// TIA Portal project "2022.04.30-电机顺启" (V17)

(* hardware
DEVICE "S7-1500/ET200MP station_1"  S7-1500 station
   slot 0: "导轨_0"  Rack  6ES7 590-1***0-0AA0
   slot 1: "PLC_1"  CPU 1516-3 PN/DP  6ES7 516-3AN00-0AB0  V1.7
      slot 3: "CPU 显示_1"  6ES7591-1BA00-0AA0
      slot 32768: "PROFINET 接口_1"  X1
         slot 32769: "端口_1"  X1 P1
         slot 32770: "端口_2"  X1 P2
      slot 33024: "PROFINET 接口_2"  X2
         slot 33025: "端口_1"  X2 P1
      slot 33280: "DP 接口_1"  X3
   slot 2: "DI 32x24VDC BA_1"  DI 32x24VDC BA  6ES7 521-1BL10-0AA0  V1.1
   slot 3: "DQ 32x24VDC/0.5A HF_1"  DQ 32x24VDC/0.5A HF  6ES7 522-1BL01-0AB0  V1.1
*)

// ===== PLC "PLC_1"  CPU 1516-3 PN/DP =====

VAR_GLOBAL   // PLC tag table "默认变量表"
   "启动按钮" AT %I0.0 : Bool;
   "停止按钮" AT %I0.1 : Bool;
   "复位按钮" AT %I0.2 : Bool;
   "按钮4" AT %I0.3 : Bool;
   "按钮5" AT %I0.4 : Bool;
   "按钮6" AT %I0.5 : Bool;
   "按钮7" AT %I0.6 : Bool;
   "按钮8" AT %I0.7 : Bool;
   "按钮9" AT %I1.0 : Bool;
   "按钮10" AT %I1.1 : Bool;
   "按钮11" AT %I1.2 : Bool;
   "电机A" AT %Q0.0 : Bool;
   "电机B" AT %Q0.1 : Bool;
   "电机C" AT %Q0.2 : Bool;
   "闪烁指示灯" AT %Q0.3 : Bool;
   "指示灯5" AT %Q0.4 : Bool;
   "指示灯6" AT %Q0.5 : Bool;
   "指示灯7" AT %Q0.6 : Bool;
   "指示灯8" AT %Q0.7 : Bool;
   "指示灯9" AT %Q1.0 : Bool;
   "指示灯10" AT %Q1.1 : Bool;
   "指示灯11" AT %Q1.2 : Bool;
   "指示灯12" AT %Q1.3 : Bool;
   "Clock_Byte" AT %MB0 : Byte;
   "Clock_10Hz" AT %M0.0 : Bool;
   "Clock_5Hz" AT %M0.1 : Bool;
   "Clock_2.5Hz" AT %M0.2 : Bool;
   "Clock_2Hz" AT %M0.3 : Bool;
   "Clock_1.25Hz" AT %M0.4 : Bool;
   "Clock_1Hz" AT %M0.5 : Bool;
   "Clock_0.625Hz" AT %M0.6 : Bool;
   "Clock_0.5Hz" AT %M0.7 : Bool;
   "停止" AT %M2.0 : Bool;
   "Tag_2" AT %M3.0 : Bool;
   "电机B停止" AT %M2.1 : Bool;
   "电机A停止" AT %M2.2 : Bool;
   "1" AT %M1.0 : Bool;
   "0" AT %M1.1 : Bool;
END_VAR

DATA_BLOCK "定时器"   // DB1
{ S7_Optimized_Access := 'TRUE' }
VERSION : 0.1
   VAR
      电机B启动 : IEC_TIMER;
      电机C启动 : IEC_TIMER;
      电机B停止 : IEC_TIMER;
      电机A停止 : IEC_TIMER;
   END_VAR
BEGIN
END_DATA_BLOCK

FUNCTION "电机启动顺停LAD" : Void   // FC1, LAD
{ S7_Optimized_Access := 'TRUE' }
VERSION : 0.1
BEGIN

REGION Network 1: 电机A启动
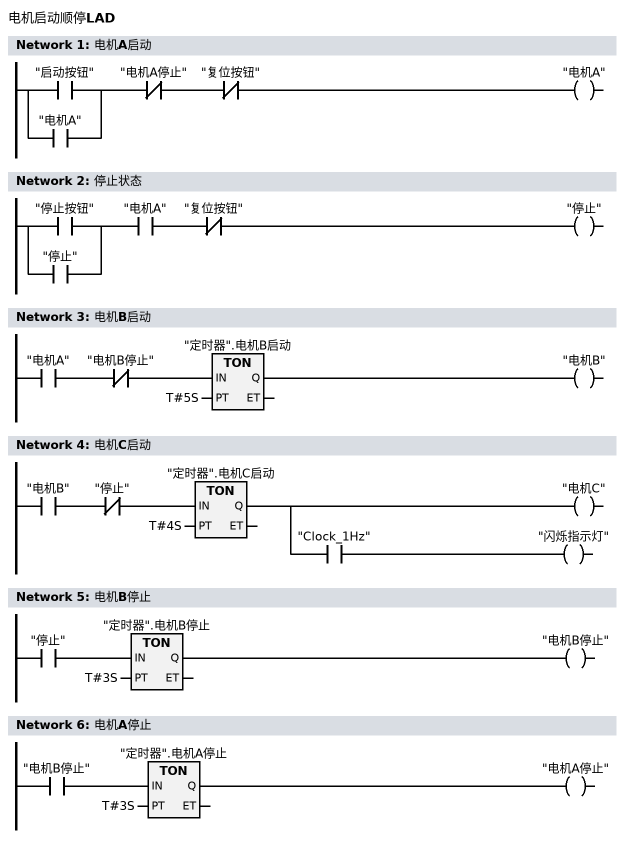
   RUNG wire#powerrail
      Contact( "启动按钮" )
      wire#w1
      I_Contact( "电机A停止" )
      I_Contact( "复位按钮" )
      Coil( "电机A" )
   END_RUNG
   RUNG wire#powerrail
      Contact( "电机A" )
   END_RUNG wire#w1
   // the same network as SCL:
   "电机A" := ("启动按钮" OR "电机A") AND NOT "电机A停止" AND NOT "复位按钮";
END_REGION

REGION Network 2: 停止状态
   RUNG wire#powerrail
      Contact( "停止按钮" )
      wire#w1
      Contact( "电机A" )
      I_Contact( "复位按钮" )
      Coil( "停止" )
   END_RUNG
   RUNG wire#powerrail
      Contact( "停止" )
   END_RUNG wire#w1
   // the same network as SCL:
   "停止" := ("停止按钮" OR "停止") AND "电机A" AND NOT "复位按钮";
END_REGION

REGION Network 3: 电机B启动
   "定时器".电机B启动.TON(IN := "电机A" AND NOT "电机B停止", PT := T#5S);
   "电机B" := "定时器".电机B启动.Q;
END_REGION

REGION Network 4: 电机C启动
   "定时器".电机C启动.TON(IN := "电机B" AND NOT "停止", PT := T#4S);
   "电机C" := "定时器".电机C启动.Q;
   "闪烁指示灯" := "定时器".电机C启动.Q AND "Clock_1Hz";
END_REGION

REGION Network 5: 电机B停止
   "定时器".电机B停止.TON(IN := "停止", PT := T#3S);
   "电机B停止" := "定时器".电机B停止.Q;
END_REGION

REGION Network 6: 电机A停止
   "定时器".电机A停止.TON(IN := "电机B停止", PT := T#3S);
   "电机A停止" := "定时器".电机A停止.Q;
END_REGION
END_FUNCTION

FUNCTION "顺序启动FBD" : Void   // FC2, FBD
{ S7_Optimized_Access := 'TRUE' }
VERSION : 0.1
BEGIN

REGION Network 1
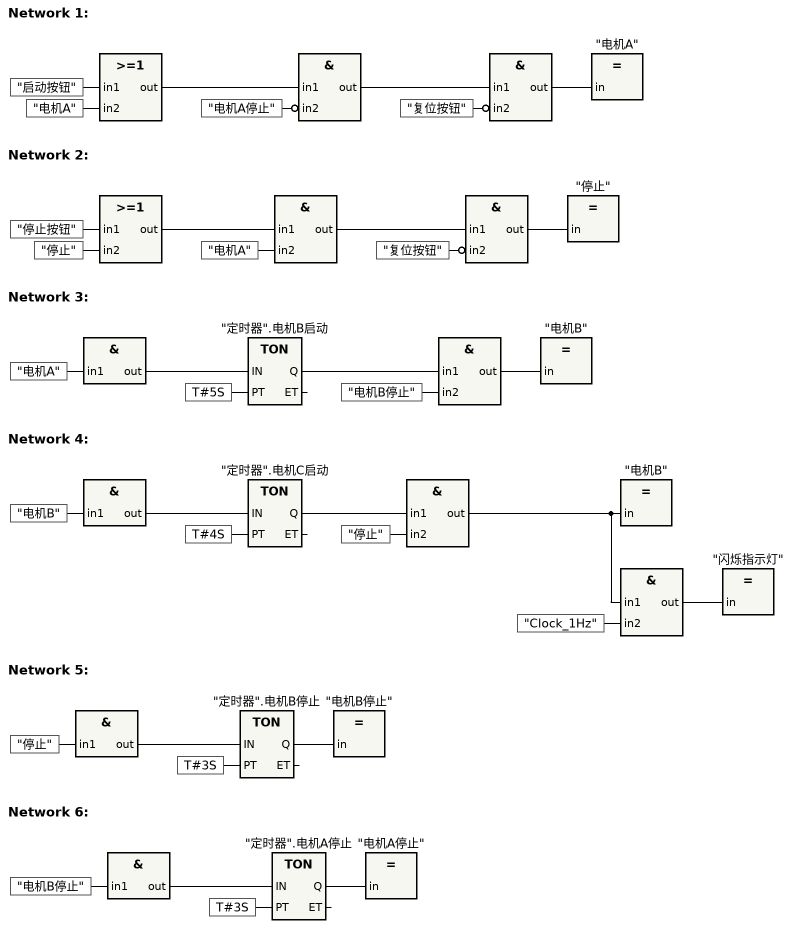
   "电机A" := ("启动按钮" OR "电机A") AND NOT "电机A停止" AND NOT "复位按钮";
END_REGION

REGION Network 2
   "停止" := ("停止按钮" OR "停止") AND "电机A" AND NOT "复位按钮";
END_REGION

REGION Network 3
   "定时器".电机B启动.TON(IN := "电机A", PT := T#5S);
   "电机B" := "定时器".电机B启动.Q AND "电机B停止";
END_REGION

REGION Network 4
   "定时器".电机C启动.TON(IN := "电机B", PT := T#4S);
   "电机B" := "定时器".电机C启动.Q AND "停止";
   "闪烁指示灯" := "电机B" AND "Clock_1Hz";
END_REGION

REGION Network 5
   "定时器".电机B停止.TON(IN := "停止", PT := T#3S);
   "电机B停止" := "定时器".电机B停止.Q;
END_REGION

REGION Network 6
   "定时器".电机A停止.TON(IN := "电机B停止", PT := T#3S);
   "电机A停止" := "定时器".电机A停止.Q;
END_REGION
END_FUNCTION

FUNCTION "电机顺序启停SCL" : Void   // FC3, SCL
{ S7_Optimized_Access := 'TRUE' }
VERSION : 0.1
BEGIN
   //电机A启动
   IF "启动按钮" = TRUE THEN
       "电机A停止" := 1;
   END_IF;
   IF "电机A" = TRUE OR "复位按钮" = TRUE THEN
       "电机A" := 0;
   END_IF;

   //停止状态
   IF "停止按钮" = TRUE THEN
       "停止" := 1;
   END_IF;
   IF "电机A" = FALSE OR "复位按钮" = TRUE THEN
       "停止" := 0;
   END_IF;
   //电机B启动
   IF "电机B停止"=FALSE THEN
       "定时器".电机B启动.TON(IN := "电机A",
                       PT := T#5S,
                       Q => "电机B"
       );
   END_IF;
   ELSE 
       "电机B" := FALSE;
   //电机C启动
   IF "停止" = FALSE THEN
       "定时器".电机C启动.TON(IN := "电机B",
                       PT := T#5S,
                       Q => "电机C"
       );
   END_IF;
   ELSE
       "电机C" := FALSE;

   //电机B停止
   IF "停止" = FALSE THEN
       "定时器".电机B停止.TON(IN := "停止",
                       PT := T#5S,
                       Q => "电机B停止"
       );
   END_IF;

   //电机A停止
   IF "电机B停止" = FALSE THEN
       "定时器".电机A停止.TON(IN := "电机B停止",
                       PT := T#3S,
                       Q => "电机A停止"
       );
   END_IF;

   //指示灯闪烁
   IF "电机C"  THEN
       "闪烁指示灯"：=TRUE；
   END_IF;
END_FUNCTION

ORGANIZATION_BLOCK "Main"   // OB1, LAD, ProgramCycle
TITLE = "Main Program Sweep (Cycle)"
{ S7_Optimized_Access := 'TRUE' }
VERSION : 0.1
   VAR_INPUT
      Initial_Call : Bool;   // Initial call of this OB
      Remanence : Bool;   // =True, if remanent data are available
   END_VAR
BEGIN

REGION Network 1: 1
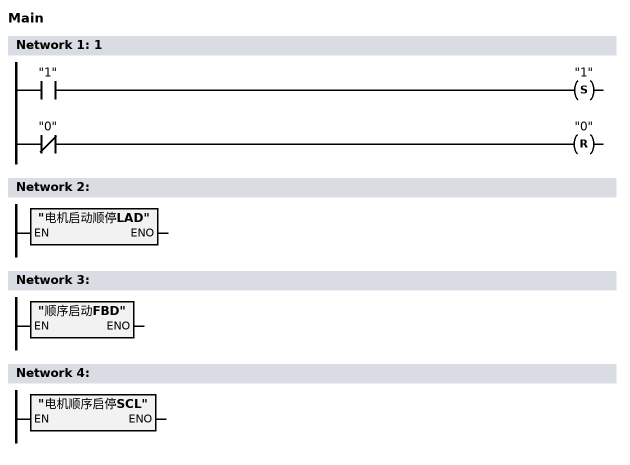
   RUNG wire#powerrail
      Contact( "1" )
      S_Coil( "1" )
   END_RUNG
   RUNG wire#powerrail
      I_Contact( "0" )
      R_Coil( "0" )
   END_RUNG
   // the same network as SCL:
   IF "1" THEN "1" := TRUE; END_IF;
   IF NOT "0" THEN "0" := FALSE; END_IF;
END_REGION

REGION Network 2
   RUNG wire#powerrail
      "电机启动顺停LAD"()
   END_RUNG
   // the same network as SCL:
   "电机启动顺停LAD"();
END_REGION

REGION Network 3
   RUNG wire#powerrail
      "顺序启动FBD"()
   END_RUNG
   // the same network as SCL:
   "顺序启动FBD"();
END_REGION

REGION Network 4
   RUNG wire#powerrail
      "电机顺序启停SCL"()
   END_RUNG
   // the same network as SCL:
   "电机顺序启停SCL"();
END_REGION
END_ORGANIZATION_BLOCK